{attribute 'linkalways'} 
{attribute 'no_explicit_call' := 'This FB is a CLASS and must be accessed using methods or properties'}
{attribute 'enable_dynamic_creation'}
FUNCTION_BLOCK FINAL LT_INT EXTENDS Node
VAR
	in1 : _INT(0);
	in2 : _INT(0);
	out : _BOOL(FALSE);
END_VAR

METHOD PUBLIC Clone : I_Node
VAR
	pNode : POINTER TO LT_INT;
END_VAR
pNode := __NEW(LT_INT);
Clone := pNode^;
END_METHOD

METHOD FB_init : BOOL
VAR_INPUT
	bInitRetains : BOOL; // if TRUE, the retain variables are initialized (warm start / cold start)
	bInCopyCode : BOOL;  // if TRUE, the instance afterwards gets moved into the copy code (online change)
END_VAR
AddInput('in1',THIS^.in1);
AddInput('in2',THIS^.in2);
AddOutput('out', THIS^.out);
END_METHOD

METHOD PROTECTED OnExecute
VAR
END_VAR
out.Value := in1.Value < in2.Value;
END_METHOD

END_FUNCTION_BLOCK

(* stored: Version 1.1.0.1, ProductVersion 3.1.4024.15
   POU LT_INT: Id {3a0994c7-ea0d-44e5-9989-2d66ea094fed}, SpecialFunc None
   Folder Constructor: Id {97cabcb1-6ff8-431d-9f60-31bd9e35e164}
   Method Clone: Id {d932eb4d-f6a0-4711-85bc-0fb71ac4ca2d}
   Method FB_init: Id {c06b1039-bbd4-4d60-8f66-d99c6d5b310d}
   Method OnExecute: Id {c09453a5-306a-4c8e-9e2e-05dd1a79997b} *)
